{attribute 'qualified_only'}
{attribute 'strict'}
(*
Some NC Error codes

Source: https://infosys.beckhoff.com/content/1033/tc3ncerrcode/1521556875.html?id=2911757239699425890
*)
TYPE NcErrorCodes : (
    CONTROLLER_ERROR_CONTROLLER_ID_NOT_ALLOWED := 17664,
    CONTROLLER_ERROR_CONTROLLER_TYPE_NOT_ALLOWED := 17665,
    CONTROLLER_ERROR_OPERATION_MODE_CONTROLLER_NOT_ALLOWED := 17666,
    CONTROLLER_ERROR_WEIGHTING_OF_THE_VELOCITY_PRE_CONTROL_NOT_ALLOWED := 17667,
    CONTROLLER_ERROR_LAG_ERROR_MONITOR_POSITION_NOT_ALLOWED := 17668,
    CONTROLLER_ERROR_LAG_MONITORING_VELOCITY_NOT_ALLOWED := 17669,
    CONTROLLER_ERROR_LAG_ERROR_WINDOW_POSITION_NOT_ALLOWED := 17670,
    CONTROLLER_ERROR_LAG_ERROR_FILTER_TIME_POSITION_NOT_ALLOWED := 17671,
    CONTROLLER_ERROR_LAG_ERROR_WINDOW_VELOCITY_NOT_ALLOWED := 17672,
    CONTROLLER_ERROR_LAG_ERROR_FILTER_TIME_VELOCITY_NOT_ALLOWED := 17673,
    CONTROLLER_ERROR_CONTROLLER_OUTPUT_LIMITATION_OUTPUT_LIMITATION_NOT_ALLOWED := 17674,
    CONTROLLER_ERROR_PROPORTIONAL_GAIN_KV_OR_KP_CONTROLLER_NOT_ALLOWED := 17680,
    CONTROLLER_ERROR_INTEGRAL_ACTION_TIME_TN_CONTROLLER_NOT_ALLOWED_POSITION := 17681,
    CONTROLLER_ERROR_RATE_TIME_TV_CONTROLLER_NOT_ALLOWED_POSITION := 17682,
    CONTROLLER_ERROR_DAMPING_TIME_TD_CONTROLLER_NOT_ALLOWED_POSITION := 17683,
    CONTROLLER_ERROR_ACTIVATION_OF_THE_AUTOMATIC_OFFSET_CALIBRATION_NOT_ALLOWED := 17684,
    CONTROLLER_ERROR_ADDITIONAL_PROPORTIONAL_GAIN_KV_OR_KP_CONTROLLER_NOT_ALLOWED := 17685,
    CONTROLLER_ERROR_REFERENCE_VELOCITY_FOR_ADDITIONAL_PROP_GAIN_CONTROLLER_NOT_ALLOWED := 17686,
    CONTROLLER_ERROR_PROPORTIONAL_GAIN_PA_PROPORTION_NOT_ALLOWED := 17687,
    CONTROLLER_ERROR_PROPORTIONAL_GAIN_KV_CONTROLLER_NOT_ALLOWED := 17688,
    CONTROLLER_ERROR_INTEGRAL_ACTION_TIME_TN_CONTROLLER_NOT_ALLOWED_VELOCITY := 17689,
    CONTROLLER_ERROR_VELOCITY_FILTER_TIME_NOT_ALLOWED := 17692,
    CONTROLLER_ERROR_DEAD_RANGE_NOT_ALLOWED := 17693,
    CONTROLLER_ERROR_PROPORTIONAL_GAIN_KCP_NOT_ALLOWED := 17695,
    CONTROLLER_ERROR_RATE_TIME_TV_CONTROLLER_NOT_ALLOWED := 17696,
    CONTROLLER_ERROR_DAMPING_TIME_TD_CONTROLLER_NOT_ALLOWED := 17697,
    CONTROLLER_ERROR_LIMITATION_OF_THE_I_PART_NOT_ALLOWED := 17698,
    CONTROLLER_ERROR_LIMITATION_OF_THE_D_PART_NOT_ALLOWED := 17699,
    CONTROLLER_ERROR_PARAMETER_DEACTIVATION_OF_THE_I_PART_DURING_TRAVEL_NOT_ALLOWED := 17700,
    CONTROLLER_ERROR_PARAMETER_FILTER_TIME_FOR_P_T2_FILTER_NOT_ALLOWED := 17701,
    CONTROLLER_ERROR_VELOCITY_OBSERVER_PARAMETERIZED_MODE_IS_NOT_ALLOWED := 17702,
    CONTROLLER_ERROR_VELOCITY_OBSERVER_MOTOR_TORQUE_CONSTANT_KT_OR_KF_IS_NOT_ALLOWED := 17703,
    CONTROLLER_ERROR_VELOCITY_OBSERVER_MOTOR_MOMENT_OF_INERTIA_JM_IS_NOT_ALLOWED := 17704,
    CONTROLLER_ERROR_VELOCITY_OBSERVER_BANDWIDTH_F0_IS_NOT_ALLOWED := 17705,
    CONTROLLER_ERROR_VELOCITY_OBSERVER_CORRECTION_FACTOR_KC_IS_NOT_ALLOWED := 17706,
    CONTROLLER_ERROR_VELOCITY_OBSERVER_TIME_CONSTANT_T_FOR_1ST_ORDER_FILTER_NOT_ALLOWED := 17707,
    CONTROLLER_ERROR_VELOCITY_OBSERVER_AMPLITUDE_DAMPING_FOR_2ND_ORDER_FILTER_NOT_ALLOWED := 17708,
    CONTROLLER_ERROR_VELOCITY_OBSERVER_FREQUENCY_FOR_2ND_ORDER_FILTER_NOT_ALLOWED := 17709,
    CONTROLLER_ERROR_CONTROLLER_INITIALIZATION := 17728,
    CONTROLLER_ERROR_AXIS_ADDRESS := 17729,
    CONTROLLER_ERROR_DRIVE_ADDRESS := 17730,
    CONTROLLER_ERROR_LAG_ERROR_MONITOR_POSITION := 17744,
    CONTROLLER_ERROR_LAG_MONITORING_VELOCITY := 17745,
    CONTROLLER_ERROR_INTERNAL_ERROR_CONTROLERR_RANGE_AREA_ASIDE := 17824,
    CONTROLLER_ERROR_INTERNAL_ERROR_CONTROLERR_RANGE_AREA_BSIDE := 17825,
    CONTROLLER_ERROR_INTERNAL_ERROR_CONTROLERR_RANGE_QNENN := 17826,
    CONTROLLER_ERROR_INTERNAL_ERROR_CONTROLERR_RANGE_PNENN := 17827,
    CONTROLLER_ERROR_INTERNAL_ERROR_CONTROLERR_RANGE_AXISIDPRESP0 := 17828
);
END_TYPE

(* stored: Version 1.1.0.1
   DUT NcErrorCodes: Id {4a2189ab-d0dd-07c8-117c-3fab1f036fcf} *)
